PROGRAM AuxiliaryControl
VAR
	// start delay for the dehumidifier to prevent overcurrent
	DeHumidifierDelay:	TON;
	DeHumidifier:		BOOL;
END_VAR
VAR CONSTANT
	humidity_high:	REAL := 75.0;
	humidity_low:	REAL := 65.0;
END_VAR

// turn off dehumidifier if dome is open
IF Environment.HumidityDome >= humidity_high AND DomeControl.DomeClosed THEN
	DeHumidifier := TRUE;
ELSIF Environment.HumidityDome < humidity_low OR DomeControl.DomeOpened OR Environment.Humidity < Environment.HumidityDome THEN
	DeHumidifier := FALSE;
END_IF

// delay startup of the dehumidifier to prevent power-spike
DeHumidifierDelay(IN := DeHumidifier, PT := T#5S, Q=> GVL_Dome.DeHumidifier);

END_PROGRAM

(* stored: Version 1.1.0.1, ProductVersion 3.1.4024.9
   POU AuxiliaryControl: Id {30a3eb2e-ebab-4f9f-a38d-cee5e71b2e38}, SpecialFunc None *)
